(* CoDeSys 2.3 library: VectorLibrary.lib *)
(* Libraries: oscat_basic_333.lib 24.4.18 10:21:04 *)

(* POU PLC_PRG, ST *)
PROGRAM PLC_PRG
VAR
END_VAR

END_PROGRAM
